SUBAPPLICATION Ventilsteuerung_Uebung_020a (* DigitalInput_I1 auf DigitalOutput_Q1 *)
  (* Standard: 61499-2 *)
  (* Version 1.0, 2023-10-23, franz *)
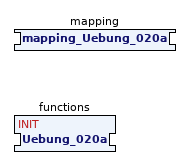
  SUBAPPS
    mapping : mapping_Uebung_020a;
    functions : Uebung_020a;
  END_SUBAPPS
END_SUBAPPLICATION
